FUNCTION_BLOCK CamModule EXTENDS FB_PackML_BaseModule
VAR
	CamShaft	  : FB_Component_BasicAxis	  := (Name := 'Cam Shaft');
	CamFollower	  : FB_Component_CamSlaveAxis := (Name := 'Cam Follower');
	CamParameters : ST_CamParameters;
	HMI			  : ST_EM_HMI;
END_VAR

METHOD PROTECTED Aborting
VAR
	CamShaftStop	: BOOL;
	CamFollowerStop : BOOL;
END_VAR
// Mode is ignored
CASE SequenceState OF
	0:
		NoStateTasksToComplete := FALSE;
		SequenceState		   := SequenceState + 10;

		// Setting Override to 100 will ensure velocity calculations are not limited
		CamShaft.Override	 := 100;
		CamFollower.Override := 100;

		// The below code is used to call the stop method of each axis while still in State 0, this is done for efficeniceny while aborting.

		// Stop all Axes
		CamShaftStop	:= CamShaft.Stop() OR CamShaft.Error;
		CamFollowerStop := CamFollower.Stop() OR CamFollower.Error;
		IF CamShaftStop AND CamFollowerStop THEN
			SequenceState := SequenceState + 10;
		END_IF

	10:
		IF CamShaft.Stopped AND CamFollower.Stopped THEN
			SequenceState := SequenceState + 10;
		END_IF

	20: // Disable Axis
		IF CamShaft.Disable() THEN
			SequenceState := SequenceState + 10;
		END_IF

	30:
		IF CamFollower.Disable() THEN
			SequenceState := SequenceState + 10;
		END_IF

	40:
		IF NOT CamShaft.Enabled AND NOT CamFollower.Enabled THEN
			SequenceState := SequenceState + 10;
		END_IF

	50:
		StateTasksComplete := TRUE;
END_CASE

SUPER^.Aborting();
END_METHOD

// This method contains code which will execute when this PackML module is in the Clearing state
METHOD PROTECTED Clearing

// Note: The Clear command can also be thought of as a fault reset depite the ambiguity in the naming of the Reset state. 

// This method is called as required by StateControl()
// Mode is ignored
CASE SequenceState OF
	0:
		NoStateTasksToComplete := FALSE;
		SequenceState		   := SequenceState + 10;

	10: // Reset Axis if Error
		IF CamShaft.Error THEN
			IF CamShaft.Reset() THEN
				SequenceState := SequenceState + 10;
			END_IF
		ELSE
			SequenceState := SequenceState + 10;
		END_IF

	20:
		IF CamFollower.InSync THEN
			IF CamFollower.Stop() THEN // This is used to decouple the axis
				SequenceState := SequenceState + 10;
			END_IF
		ELSE
			SequenceState := SequenceState + 10;
		END_IF

	30:
		IF CamFollower.Error THEN
			IF CamFollower.Reset() THEN
				SequenceState := SequenceState + 10;
			END_IF
		ELSE
			SequenceState := SequenceState + 10;
		END_IF

	40:
		StateTasksComplete := TRUE;
END_CASE

SUPER^.Clearing();
END_METHOD

METHOD PROTECTED Completing
CASE SequenceState OF
	0:
		NoStateTasksToComplete := FALSE;
		SequenceState		   := SequenceState + 10;

	10:
		IF CamShaft.Stop() THEN // This will also GearOut
			SequenceState := SequenceState + 10;
		END_IF

	20:
		IF CamFollower.Stop() THEN // This will also GearOut
			SequenceState := SequenceState + 10;
		END_IF

	30:
		IF CamShaft.Stopped AND CamFollower.Stopped THEN
			SequenceState := SequenceState + 10;
		END_IF

	40:
		StateTasksComplete := TRUE;
END_CASE

SUPER^.Completing();
END_METHOD

// This method serves as the entry point for all underlying FB logic

// This method should be called cyclically by descendant function blocks by invoking SUPER^.CyclicLogic().  Alternatively, the contents of this method could be reimplemented entirely in which case a call to this method would not be necessary.
METHOD PUBLIC CyclicLogic
IF NOT _InitComplete THEN
	_InitComplete := Initialize();
	RETURN;
END_IF

// HMI Status Update
HMI.Sts.CurrentTable := CamFollower.RunningTable;

// Change Activation Mode
IF HMI.Cmd.ChangeMode THEN
	CASE HMI.Cfg.CamActivationMode OF
		0:
			CamParameters.ChangeOptions.ActivationMode := MC_CamActivationMode.MC_CAMACTIVATION_NEXTCYCLE;

		1:
			CamParameters.ChangeOptions.ActivationMode := MC_CamActivationMode.MC_CAMACTIVATION_ASSOONASPOSSIBLE;
	END_CASE

	IF CamFollower.ChangeMode() THEN
		HMI.Cmd.ChangeMode := FALSE;
	END_IF
END_IF

SUPER^.CyclicLogic();
END_METHOD

// This method contains code which will execute when this PackML module is in the Execute state
METHOD PROTECTED Execute

(*
The base implementation of this method is empty. User must override this method to provide functionality.
This method is called as required by StateControl()
*)
CASE _CurrentMode OF
	E_PMLUnitMode.ePMLUnitMode_Production:
		CASE SequenceState OF
			0: // Start Cam Shaft
				IF CamShaft.MoveVelocity(50.0, FALSE) THEN
					SequenceState := SequenceState + 10;
				END_IF

			10: // Checking that the Cam Shaft is near the commanded speed 
				IF (CamShaft.ActualVelocity > (CamShaft.SetVelocity * 0.9)) THEN
					SequenceState := SequenceState + 10;
				END_IF

			20:
				IF HMI.Cmd.ChangeTable THEN
					HMI.Cmd.ChangeTable := FALSE;
					CASE CamFollower.RunningTable OF
						1:
							CamFollower.CamParameters.CamTableId  := 1;
							CamFollower.CamParameters.TableSelect := 2;

						2:
							CamFollower.CamParameters.CamTableId  := 1;
							CamFollower.CamParameters.TableSelect := 1;
					END_CASE

					SequenceState := SequenceState + 10;
				END_IF

			30:
				IF CamFollower.RunningTable = CamFollower.CamParameters.TableSelect THEN
					SequenceState := 20;
				END_IF;
		END_CASE
END_CASE
END_METHOD

// Basic module initialization logic
METHOD PROTECTED Initialize : BOOL;

// This method is called by CyclicLogic() as required
Initialize := FALSE;
CASE DescendantSequenceState OF
	0:
		RegisterComponent(Component := CamShaft);
		RegisterComponent(Component := CamFollower);
		DescendantSequenceState := DescendantSequenceState + 10;

	10:
		IF SUPER^.Initialize() THEN
			DescendantSequenceState := DescendantSequenceState + 10;
		END_IF

	20:
		// Create the Cam table data and store in CamParameters
		WriteCamParameters();

		// Replace the default value of MC_CAMACTIVATION_INSTANTANEOUS with MC_CAMACTIVATION_NEXTCYCLE
		CamParameters.CamInOptions.ActivationMode  := MC_CamActivationMode.MC_CAMACTIVATION_NEXTCYCLE;
		CamParameters.ChangeOptions.ActivationMode := MC_CamActivationMode.MC_CAMACTIVATION_NEXTCYCLE;

		// Set the Reference for the Axis Cam Parameters to the CamParameters
		CamFollower.CamParameters REF= CamParameters;

		// Setting the Reference of the FB_Component_CamSlaveAxis must be done after the component has been initialized
		CamFollower.Master REF= CamShaft.Axis;

		//
		DescendantSequenceState := DescendantSequenceState + 10;

	30:
		Initialize := TRUE;
END_CASE
END_METHOD

METHOD PROTECTED Starting
CASE _CommandedMode OF
	ePMLProtUnitMode_Production:
		CASE SequenceState OF
			0:
				NoStateTasksToComplete := FALSE;
				SequenceState		   := SequenceState + 10;

			10: // Enable Axis 
				IF CamShaft.Enable() THEN
					SequenceState := SequenceState + 10;
				END_IF

			20:
				IF CamShaft.Enabled THEN
					SequenceState := SequenceState + 10;
				END_IF

			30: // This step is not required, but is used in this demo to ensure the CamShaft starts at 0
				IF CamShaft.MoveModulo(0.0, MC_Direction.MC_Shortest_Way, 0) THEN
					SequenceState := SequenceState + 10;
				END_IF

			40:
				IF NOT CamShaft.Busy THEN
					IF NOT CamShaft.Error THEN
						SequenceState := SequenceState + 10;
					END_IF
				END_IF

			50: // Enable Axis
				IF CamFollower.Enable() THEN
					SequenceState := SequenceState + 10;
				END_IF

			60:
				IF CamFollower.Enabled THEN
					SequenceState := SequenceState + 10;
				END_IF

			70: // This step is not required, but is used in the demo to ensure the follower starts at 0
				IF CamFollower.MoveAbsolute(0, 0) THEN
					SequenceState := SequenceState + 10;
				END_IF

			80:
				IF NOT CamFollower.Busy THEN
					IF NOT CamFollower.Error THEN
						SequenceState := SequenceState + 10;
					END_IF
				END_IF

			90: // Verify the Master axis is ready 
				IF CamFollower.Master.Status.Operational THEN
					SequenceState := SequenceState + 10;
				END_IF

			100: // Select the Cam Table to be used
				CamFollower.CamParameters.CamTableId  := 1;
				CamFollower.CamParameters.TableSelect := 1;
				SequenceState						  := SequenceState + 10;

			110: // Couple to Cam table with Master axis
				IF CamFollower.WaitingForCommand THEN
					IF CamFollower.StartSync() THEN // The Start Sync command will move the axes tho the necessary positions and then CamIn
						SequenceState := SequenceState + 10;
					END_IF
				END_IF

			120:
				IF CamFollower.InSync THEN
					SequenceState := SequenceState + 10;
				END_IF

			130:
				StateTasksComplete := TRUE;
		END_CASE
END_CASE

SUPER^.Starting();
END_METHOD

METHOD PROTECTED Stopping
CASE SequenceState OF
	0:
		NoStateTasksToComplete := FALSE;
		SequenceState		   := SequenceState + 10;

	10:
		IF CamShaft.Stop() THEN // This will also GearOut 
			SequenceState := SequenceState + 10;
		END_IF

	20:
		IF CamFollower.Stop() THEN // This will also GearOut  
			SequenceState := SequenceState + 10;
		END_IF

	30:
		IF CamShaft.Stopped AND CamFollower.Stopped THEN
			SequenceState := SequenceState + 10;
		END_IF

	40:
		StateTasksComplete := TRUE;
END_CASE

SUPER^.Stopping();
END_METHOD

METHOD WriteCamParameters
VAR
	PointIdx : UDINT;
	i		 : UDINT;
	Start	 : UDINT;
END_VAR
// Table 1 Data
CamParameters.CamTableId										:= 1;
CamParameters.CamTable[CamParameters.CamTableId].NumberOfPoints := Parameters_MotionControl.CAM_SLAVE_AXIS_MAX_CAM_POINTS;
PointIdx														:= 0;

//
PointIdx																			:= PointIdx + 1;
CamParameters.CamTable[CamParameters.CamTableId].Points[PointIdx].PointIndex		:= PointIdx;
CamParameters.CamTable[CamParameters.CamTableId].Points[PointIdx].FunctionType		:= MC_MotionFunctionType.MOTIONFUNCTYPE_POLYNOM5;
CamParameters.CamTable[CamParameters.CamTableId].Points[PointIdx].PointType			:= MC_MotionPointType.MOTIONPOINTTYPE_REST;
CamParameters.CamTable[CamParameters.CamTableId].Points[PointIdx].RelIndexNextPoint := 1;
CamParameters.CamTable[CamParameters.CamTableId].Points[PointIdx].MasterPos			:= 0.0;
CamParameters.CamTable[CamParameters.CamTableId].Points[PointIdx].SlavePos			:= 0.0;

//
PointIdx																			:= PointIdx + 1;
CamParameters.CamTable[CamParameters.CamTableId].Points[PointIdx].PointIndex		:= PointIdx;
CamParameters.CamTable[CamParameters.CamTableId].Points[PointIdx].FunctionType		:= MC_MotionFunctionType.MOTIONFUNCTYPE_POLYNOM5;
CamParameters.CamTable[CamParameters.CamTableId].Points[PointIdx].PointType			:= MC_MotionPointType.MOTIONPOINTTYPE_VELOCITY;
CamParameters.CamTable[CamParameters.CamTableId].Points[PointIdx].RelIndexNextPoint := 1;
CamParameters.CamTable[CamParameters.CamTableId].Points[PointIdx].MasterPos			:= 90.0;
CamParameters.CamTable[CamParameters.CamTableId].Points[PointIdx].SlavePos			:= 10.0;

//
PointIdx																			:= PointIdx + 1;
CamParameters.CamTable[CamParameters.CamTableId].Points[PointIdx].PointIndex		:= PointIdx;
CamParameters.CamTable[CamParameters.CamTableId].Points[PointIdx].FunctionType		:= MC_MotionFunctionType.MOTIONFUNCTYPE_POLYNOM5;
CamParameters.CamTable[CamParameters.CamTableId].Points[PointIdx].PointType			:= MC_MotionPointType.MOTIONPOINTTYPE_VELOCITY;
CamParameters.CamTable[CamParameters.CamTableId].Points[PointIdx].RelIndexNextPoint := 1;
CamParameters.CamTable[CamParameters.CamTableId].Points[PointIdx].MasterPos			:= 270.0;
CamParameters.CamTable[CamParameters.CamTableId].Points[PointIdx].SlavePos			:= 0.0;

// Fill the rest of the table with ignore points
Start := PointIdx + 1;
FOR PointIdx := Start TO Parameters_MotionControl.CAM_SLAVE_AXIS_MAX_CAM_POINTS DO
	CamParameters.CamTable[CamParameters.CamTableId].Points[PointIdx].PointIndex		:= PointIdx;
	CamParameters.CamTable[CamParameters.CamTableId].Points[PointIdx].FunctionType		:= MC_MotionFunctionType.MOTIONFUNCTYPE_NOTDEF;
	CamParameters.CamTable[CamParameters.CamTableId].Points[PointIdx].PointType			:= MC_MotionPointType.MOTIONPOINTTYPE_IGNORE;
	CamParameters.CamTable[CamParameters.CamTableId].Points[PointIdx].RelIndexNextPoint := 1;
	CamParameters.CamTable[CamParameters.CamTableId].Points[PointIdx].MasterPos			:= 0.0;
	CamParameters.CamTable[CamParameters.CamTableId].Points[PointIdx].SlavePos			:= 0.0;
END_FOR

// Set Lasst Point RelNext to 0
CamParameters.CamTable[CamParameters.CamTableId].Points[Parameters_MotionControl.CAM_SLAVE_AXIS_MAX_CAM_POINTS].RelIndexNextPoint := 0;

// Table 2 Data
CamParameters.CamTableId										:= 2;
CamParameters.CamTable[CamParameters.CamTableId].NumberOfPoints := Parameters_MotionControl.CAM_SLAVE_AXIS_MAX_CAM_POINTS;
PointIdx														:= 0;

//
PointIdx																			:= PointIdx + 1;
CamParameters.CamTable[CamParameters.CamTableId].Points[PointIdx].PointIndex		:= PointIdx;
CamParameters.CamTable[CamParameters.CamTableId].Points[PointIdx].FunctionType		:= MC_MotionFunctionType.MOTIONFUNCTYPE_POLYNOM5;
CamParameters.CamTable[CamParameters.CamTableId].Points[PointIdx].PointType			:= MC_MotionPointType.MOTIONPOINTTYPE_REST;
CamParameters.CamTable[CamParameters.CamTableId].Points[PointIdx].RelIndexNextPoint := 1;
CamParameters.CamTable[CamParameters.CamTableId].Points[PointIdx].MasterPos			:= 0.0;
CamParameters.CamTable[CamParameters.CamTableId].Points[PointIdx].SlavePos			:= 0.0;

//
PointIdx																			:= PointIdx + 1;
CamParameters.CamTable[CamParameters.CamTableId].Points[PointIdx].PointIndex		:= PointIdx;
CamParameters.CamTable[CamParameters.CamTableId].Points[PointIdx].FunctionType		:= MC_MotionFunctionType.MOTIONFUNCTYPE_POLYNOM5;
CamParameters.CamTable[CamParameters.CamTableId].Points[PointIdx].PointType			:= MC_MotionPointType.MOTIONPOINTTYPE_VELOCITY;
CamParameters.CamTable[CamParameters.CamTableId].Points[PointIdx].RelIndexNextPoint := 1;
CamParameters.CamTable[CamParameters.CamTableId].Points[PointIdx].MasterPos			:= 90.0;
CamParameters.CamTable[CamParameters.CamTableId].Points[PointIdx].SlavePos			:= 20.0;

//
PointIdx																			:= PointIdx + 1;
CamParameters.CamTable[CamParameters.CamTableId].Points[PointIdx].PointIndex		:= PointIdx;
CamParameters.CamTable[CamParameters.CamTableId].Points[PointIdx].FunctionType		:= MC_MotionFunctionType.MOTIONFUNCTYPE_POLYNOM5;
CamParameters.CamTable[CamParameters.CamTableId].Points[PointIdx].PointType			:= MC_MotionPointType.MOTIONPOINTTYPE_VELOCITY;
CamParameters.CamTable[CamParameters.CamTableId].Points[PointIdx].RelIndexNextPoint := 1;
CamParameters.CamTable[CamParameters.CamTableId].Points[PointIdx].MasterPos			:= 270.0;
CamParameters.CamTable[CamParameters.CamTableId].Points[PointIdx].SlavePos			:= 20.0;

//
PointIdx																			:= PointIdx + 1;
CamParameters.CamTable[CamParameters.CamTableId].Points[PointIdx].PointIndex		:= PointIdx;
CamParameters.CamTable[CamParameters.CamTableId].Points[PointIdx].FunctionType		:= MC_MotionFunctionType.MOTIONFUNCTYPE_POLYNOM5;
CamParameters.CamTable[CamParameters.CamTableId].Points[PointIdx].PointType			:= MC_MotionPointType.MOTIONPOINTTYPE_REST;
CamParameters.CamTable[CamParameters.CamTableId].Points[PointIdx].RelIndexNextPoint := 0;
CamParameters.CamTable[CamParameters.CamTableId].Points[PointIdx].MasterPos			:= 360.0;
CamParameters.CamTable[CamParameters.CamTableId].Points[PointIdx].SlavePos			:= 0.0;

// Fill the rest of the table with ignore points
Start := PointIdx + 1;
FOR PointIdx := Start TO Parameters_MotionControl.CAM_SLAVE_AXIS_MAX_CAM_POINTS DO
	CamParameters.CamTable[CamParameters.CamTableId].Points[PointIdx].PointIndex		:= PointIdx;
	CamParameters.CamTable[CamParameters.CamTableId].Points[PointIdx].FunctionType		:= MC_MotionFunctionType.MOTIONFUNCTYPE_NOTDEF;
	CamParameters.CamTable[CamParameters.CamTableId].Points[PointIdx].PointType			:= MC_MotionPointType.MOTIONPOINTTYPE_IGNORE;
	CamParameters.CamTable[CamParameters.CamTableId].Points[PointIdx].RelIndexNextPoint := 1;
	CamParameters.CamTable[CamParameters.CamTableId].Points[PointIdx].MasterPos			:= 0.0;
	CamParameters.CamTable[CamParameters.CamTableId].Points[PointIdx].SlavePos			:= 0.0;
END_FOR

// Set Lasst Point RelNext to 0
CamParameters.CamTable[CamParameters.CamTableId].Points[Parameters_MotionControl.CAM_SLAVE_AXIS_MAX_CAM_POINTS].RelIndexNextPoint := 0;
END_METHOD

END_FUNCTION_BLOCK

(* stored: Version 1.1.0.1, ProductVersion 3.1.4024.12
   POU CamModule: Id {ddb3cd35-7a81-40ab-a1b2-be359f59229f}, SpecialFunc None
   Folder Acting States: Id {faa1328b-3dee-4665-ad83-f37760db8c73}
   Folder CyclicLogic: Id {34af7902-5adf-4564-a495-77535304ff6e}
   Method Aborting: Id {6cf75930-77b9-4f04-8720-a76f5a6fe581}
   Method Clearing: Id {9664bf73-0644-4593-adaa-3e91ecf4a27e}
   Method Completing: Id {6675e2ed-3787-4703-9a8a-227583bf4e79}
   Method CyclicLogic: Id {4ed58811-d451-469e-857f-aaceaa591767}
   Method Execute: Id {a7b0505e-11cf-49c2-93ad-d40f28ad4670}
   Method Initialize: Id {1d27b49b-eb66-4f64-a324-4b5c9edb7f49}
   Method Starting: Id {038f3a3f-7ac2-410c-9b00-0dcfd4fbb0b7}
   Method Stopping: Id {0f620c0c-c327-488f-b597-5e9ab9e0ed57}
   Method WriteCamParameters: Id {ea3ba973-03c7-4221-901d-90e5475608ee} *)
